// generates a signal build up by the specified function type. v1.4
// generates random signal (uniform, normal or chi-squared)

FUNCTION_BLOCK FB_FunctionGenerator
VAR_INPUT
	bEnable		: BOOL 	:= TRUE;
	fSamplingRate : LREAL := 10000.0; // in Hz
	nOversamples : UDINT := 10;
	fFrequency	: LREAL := 1000;	// in [Hz]
	fAmplitude	: LREAL := 1;
	fOffset		: LREAL	:= 0;	
	nDutyCycle	: UINT 	:= 50;		// % (for pulse function)
	nSeed		: INT	:= 1;	 
	aRange		: ARRAY [1..2] OF LREAL := [0,1];
	eRandType	: E_DistributionType	:= E_DistributionType.eNormal;
	eFunction	: E_FunctionType := E_FunctionType.eSine;	
END_VAR
VAR_OUTPUT
	bError		: BOOL;
	aSignal		: ARRAY[1..cOversamples] OF LREAL;
END_VAR
VAR
	bInit						: BOOL := TRUE;
	fLastSamplingRate : LREAL;
	nLastOversamples : UDINT;
	fLastFrequency				: LREAL;		// in [Hz]
	fLastAmplitude				: LREAL;
	fLastOffset					: LREAL;
	nLastDutyCycle				: UINT;
	eLastFunction				: E_FunctionType;
	
	nSamples					: UDINT;
	fCycleTime					: LREAL;		// in [s]
	fDelta						: LREAL;		// amplitude delta per sample
	fPhase						: LREAL;		// in [°]
	nSign						: INT := 1;		// 1 or -1
	fLastSignalValue			: LREAL;		// amplitude
	fPeriod						: LREAL;		// in [s]
	fAngularIncrement			: LREAL;		// in [°]
	fAngularIncrementPerCycle	: LREAL;		// in [°]
	fAngularIncrementPerSample	: LREAL;		// in [°]
	(* for modulated signal *)
	fCarrierFrequency			: LREAL := 500;	// in [Hz] (sine)
	fCarrierAmplitude			: LREAL := 1;
	fCarrierPeriod				: LREAL;		// in [s]
	fCarrierAngularIncrement			: LREAL;		// in [°]
	fCarrierAngularIncrementPerCycle	: LREAL;		// in [°]
	fCarrierAngularIncrementPerSample	: LREAL;		// in [°]
	
	fbDrand						: ARRAY[1..cOversamples] OF DRAND;		
	bNormalDist					: BOOL := TRUE;
	
	fY1							: LREAL;
	fY2							: LREAL;
	fX1							: LREAL;
	fX2							: LREAL;
	
	fbRAND1						: DRAND;
	fbRAND2						: DRAND;				
END_VAR

IF bEnable THEN

	IF fLastSamplingRate <> fSamplingRate THEN
		bInit := TRUE; // For automatic initializing
		fLastSamplingRate := fSamplingRate;
	END_IF
	IF nLastOversamples <> nOversamples THEN
		bInit := TRUE; // For automatic initializing
		nLastOversamples := nOversamples;
	END_IF
	
	IF fLastFrequency <> fFrequency THEN
		bInit := TRUE; // For automatic initializing
		fLastFrequency := fFrequency;
	END_IF
	IF fLastAmplitude <> fAmplitude THEN
		bInit := TRUE; // For automatic initializing
		fLastAmplitude := fAmplitude;
	END_IF
	IF fLastOffset <> fOffset THEN
		bInit := TRUE; // For automatic initializing
		fLastOffset := fOffset;
	END_IF
	IF nLastDutyCycle <> nDutyCycle THEN
		bInit := TRUE; // For automatic initializing
		nLastDutyCycle := nDutyCycle;
	END_IF
	IF eLastFunction <> eFunction THEN
		bInit := TRUE; // For automatic initializing
		eLastFunction := eFunction;
	END_IF
	IF bInit THEN
		// Get taks info	
//		fbGetTaskIdx();
//		fCycleTime := TwinCAT_SystemInfoVarList._TaskInfo[fbGetTaskIdx.index].CycleTime (*100ns*) / (10.0 * 1000.0 * 1000.0);	
		fCycleTime	 := nOversamples/fSamplingRate;
		fLastSignalValue := 0;
		nSign := 1;
		fAngularIncrement := 0;
		// Flush out old data
		MEMSET(ADR(aSignal), 0, SIZEOF(aSignal));
		IF fFrequency <> 0 AND fCycleTime > 0 THEN		
			// Calculate period, increments per plc cycle, increment per oversample
			IF cOversamples <> 0 THEN			
				IF eFunction = E_FunctionType.eSine THEN
					fPeriod := 1/fFrequency;
					fAngularIncrementPerCycle := 360*(fCycleTime/fPeriod);
					fAngularIncrementPerSample := fAngularIncrementPerCycle/cOversamples;
					// no phase adjustment
					bInit := FALSE;
				ELSIF eFunction = E_FunctionType.eConst	THEN
					bInit := FALSE;	
				ELSIF eFunction = E_FunctionType.eSquare	THEN
					fPeriod := 1/fFrequency;
					fAngularIncrementPerCycle := 360*(fCycleTime/fPeriod);
					fAngularIncrementPerSample := fAngularIncrementPerCycle/cOversamples;
					fPhase := 0.5*360;
					bInit := FALSE;
				ELSIF eFunction = E_FunctionType.ePulse THEN
					fPeriod := 1/fFrequency;
					fAngularIncrementPerCycle := 360*(fCycleTime/fPeriod);
					fAngularIncrementPerSample := fAngularIncrementPerCycle/cOversamples;
					IF nDutyCycle > 100 THEN
						nDutyCycle := 100;
					END_IF
					fPhase := (UDINT_TO_LREAL(nDutyCycle)/100)*360;
					bInit := FALSE;					
				ELSIF eFunction = E_FunctionType.eTriangular THEN
					fPeriod := 1/fFrequency;				
					fAngularIncrementPerCycle := 360*(fCycleTime/fPeriod);
					fAngularIncrementPerSample := fAngularIncrementPerCycle/cOversamples;
					fPhase := 0.5*360; 
					fDelta := 4*(fAmplitude/(360/fAngularIncrementPerSample));				
					bInit := FALSE;
				ELSIF eFunction = E_FunctionType.eTrapezoid THEN
					fPeriod := 1/fFrequency;				
					fAngularIncrementPerCycle := 360*(fCycleTime/fPeriod);
					fAngularIncrementPerSample := fAngularIncrementPerCycle/cOversamples;
					fPhase := 0.5*360; 
					fDelta := 4*(fAmplitude/(360/fAngularIncrementPerSample));				
					bInit := FALSE;					
				ELSIF eFunction = E_FunctionType.eSawtooth THEN
					fPeriod := 1/fFrequency;			
					fAngularIncrementPerCycle := 360*(fCycleTime/fPeriod);		
					fAngularIncrementPerSample := fAngularIncrementPerCycle/cOversamples;
					fDelta := fAmplitude/(360/fAngularIncrementPerSample);
					bInit := FALSE;
				ELSIF eFunction = E_FunctionType.eAM THEN
					fPeriod := 1/fFrequency;
					fAngularIncrementPerCycle := 360*(fCycleTime/fPeriod);
					fAngularIncrementPerSample := fAngularIncrementPerCycle/cOversamples;
					// no phase adjustment
					fCarrierPeriod := 1/fCarrierFrequency;
					fCarrierAngularIncrementPerCycle := 360*(fCycleTime/fCarrierPeriod);
					fCarrierAngularIncrementPerSample := fCarrierAngularIncrementPerCycle/cOversamples;				
					// no phase adjustment	
					bInit := FALSE;			
				ELSIF eFunction = E_FunctionType.eRand THEN	
					fbRAND1(Seed := nSeed);
					fbRAND2(Seed := nSeed+1);
					bInit := FALSE;
				ELSE
					bError := TRUE;	
				END_IF
			ELSE
				bError := TRUE;
			END_IF
		ELSE
			bError := TRUE;
		END_IF
	END_IF
	
	// Enable function generator
	IF NOT bError THEN		
		CASE eFunction OF		
			// const: constant signal
			E_FunctionType.eConst: Const();
			
			// sine: typical for vibrations originating from rotating machine
			E_FunctionType.eSine: Sine();			
			
			// square: mixed sine signals good for analyzing spectrum				
			E_FunctionType.eSquare: Square();
			
			// pulse: mixed sine signals good for analyzing spectrum				
			E_FunctionType.ePulse: Pulse();
	
			// sawtooth: ramp-type vibrations, continuously increasing			
			E_FunctionType.eSawtooth: Sawtooth();
		
			// triangular: mixed sine signals good for analyzing spectrum
			E_FunctionType.eTriangular: Triangular();
			
			// Trapezoid: trapezoid signal
			E_FunctionType.eTrapezoid: Trapezoid();
		
			// amplitude modulation: typical for vibrations originating from gear-tooth failure or bearing faults
			// Carrier signal with own frequency and amplitude		
			E_FunctionType.eAM: AM();	

			// random nosie: typical for disturbance signal				
		END_CASE
	END_IF
ELSE
	// Flush out old data
	MEMSET(ADR(aSignal), 0, SIZEOF(aSignal));
END_IF

METHOD PUBLIC AddAbsoluteNoise
VAR_INPUT
	fAbsoluteNoise	: LREAL;
END_VAR
VAR_IN_OUT
	aSignal		: ARRAY[1..cOversamples] OF LREAL;
END_VAR
VAR
	fNoise :LREAL;
END_VAR
FOR nSamples := 1 TO cOversamples DO	
	fbRAND1(Num => fNoise); // betwenn 0-1
	fNoise:= (fNoise*2 -1.0) * fAbsoluteNoise;
	aSignal[nSamples] := aSignal[nSamples] + fNoise;
END_FOR
END_METHOD

METHOD PRIVATE AM
VAR_INPUT
END_VAR
FOR nSamples := 1 TO cOversamples DO
	// base signal * carrier signal
	aSignal[nSamples] := ( fAmplitude*SIN(2*PI*(fAngularIncrement+(nSamples-1)*fAngularIncrementPerSample)/360) + fOffset )
							* ( fCarrierAmplitude*SIN(2*PI*(fCarrierAngularIncrement+(nSamples-1)*fCarrierAngularIncrementPerSample)/360) );
END_FOR
// Increment angular positions
fAngularIncrement := fAngularIncrement + fAngularIncrementPerCycle;
fCarrierAngularIncrement := fCarrierAngularIncrement + fCarrierAngularIncrementPerCycle;
END_METHOD

METHOD PRIVATE Const
VAR_INPUT
END_VAR
FOR nSamples := 1 TO cOversamples DO
	
	aSignal[nSamples] := fAmplitude;
	
	aSignal[nSamples] := aSignal[nSamples] + fOffset;
END_FOR
END_METHOD

METHOD PRIVATE Pulse
VAR_INPUT
END_VAR
FOR nSamples := 1 TO cOversamples DO
	// For pulse wave (unequal phases)
	IF (fAngularIncrement >= 360) THEN
		fAngularIncrement := fAngularIncrement - DINT_TO_LREAL(LREAL_TO_DINT(fAngularIncrement/360))*360;
		// or with Tc2_Math library: fAngularIncrement := LMOD(fAngularIncrement,360);
	END_IF
	IF (fAngularIncrement < fPhase) THEN
		nSign := 1;		
	ELSIF (fAngularIncrement >= fPhase) THEN
		nSign := 0;
	END_IF
	fAngularIncrement := fAngularIncrement + fAngularIncrementPerSample;
	
	aSignal[nSamples] := nSign*fAmplitude;
	
	aSignal[nSamples] := aSignal[nSamples] + fOffset;
END_FOR
END_METHOD

METHOD PRIVATE Sawtooth
VAR_INPUT
END_VAR
FOR nSamples := 1 TO cOversamples DO
	// For sawtooth wave (equal phase = period/2)
	IF (fAngularIncrement >= 360) THEN
		fAngularIncrement := fAngularIncrement - DINT_TO_LREAL(LREAL_TO_DINT(fAngularIncrement/360))*360;
		// or with Tc2_Math library: fAngularIncrement := LMOD(fAngularIncrement,360);
		fLastSignalValue := fLastSignalValue -fAmplitude;
	END_IF
	fAngularIncrement := fAngularIncrement + fAngularIncrementPerSample;

	aSignal[nSamples] := fLastSignalValue + fDelta;

	// Store last sample
	fLastSignalValue := aSignal[nSamples];
	
	aSignal[nSamples] := aSignal[nSamples] + fOffset;					
END_FOR
END_METHOD

METHOD PRIVATE Sine
VAR_INPUT
END_VAR
FOR nSamples := 1 TO cOversamples DO
	aSignal[nSamples] := fAmplitude*SIN(2*PI*(fAngularIncrement+(nSamples-1)*fAngularIncrementPerSample)/360);

	aSignal[nSamples] := aSignal[nSamples] + fOffset;
END_FOR

// Increment angular position
fAngularIncrement := fAngularIncrement + fAngularIncrementPerCycle;
END_METHOD

METHOD PRIVATE Square
VAR_INPUT
END_VAR
FOR nSamples := 1 TO cOversamples DO
	// For square wave (equal phase = period/2)
	IF (fAngularIncrement >= 360) THEN
		fAngularIncrement := fAngularIncrement - DINT_TO_LREAL(LREAL_TO_DINT(fAngularIncrement/360))*360;
		// or with Tc2_Math library: fAngularIncrement := LMOD(fAngularIncrement,360);
	END_IF
	IF (fAngularIncrement < fPhase) THEN
		nSign := 1;
	ELSIF (fAngularIncrement >= fPhase) THEN
		nSign := -1;
	END_IF
	fAngularIncrement := fAngularIncrement + fAngularIncrementPerSample;
	
	aSignal[nSamples] := nSign*fAmplitude;
	
	aSignal[nSamples] := aSignal[nSamples] + fOffset;
END_FOR
END_METHOD

METHOD PRIVATE Trapezoid
VAR_INPUT
END_VAR
FOR nSamples := 1 TO cOversamples DO
	IF (fAngularIncrement >= 360) THEN
		fAngularIncrement := fAngularIncrement - DINT_TO_LREAL(LREAL_TO_DINT(fAngularIncrement/360))*360;
		// or with Tc2_Math library: fAngularIncrement := LMOD(fAngularIncrement,360);
	END_IF
	// Negative delta -> Positive delta
	IF fAngularIncrement < fPhase/2 THEN	
		nSign := 1;		
	ELSIF fAngularIncrement >= fPhase/2 AND fAngularIncrement < fPhase THEN
		nSign := -1;
	ELSIF fAngularIncrement >= fPhase THEN
		nSign := 0;	
	END_IF
	fAngularIncrement := fAngularIncrement + fAngularIncrementPerSample;
	
	aSignal[nSamples] := fLastSignalValue + nSign*fDelta;
	IF aSignal[nSamples] > fAmplitude THEN
		aSignal[nSamples] := aSignal[nSamples] - 2*(aSignal[nSamples]-fAmplitude);
	ELSIF aSignal[nSamples] < (-1)*fAmplitude THEN
		aSignal[nSamples] := aSignal[nSamples] - 2*(aSignal[nSamples]+fAmplitude);
	END_IF
	
	// Store last sample
	fLastSignalValue := aSignal[nSamples];		
	
	IF fLastSignalValue > fAmplitude * 0.5 THEN
		aSignal[nSamples] := fAmplitude * 0.5;
	END_IF
	
	aSignal[nSamples] := aSignal[nSamples] + fOffset;
END_FOR
END_METHOD

METHOD PRIVATE Triangular
VAR_INPUT
END_VAR
FOR nSamples := 1 TO cOversamples DO
	IF (fAngularIncrement >= 360) THEN
		fAngularIncrement := fAngularIncrement - DINT_TO_LREAL(LREAL_TO_DINT(fAngularIncrement/360))*360;
		// or with Tc2_Math library: fAngularIncrement := LMOD(fAngularIncrement,360);
	END_IF
	// Negative delta -> Positive delta
	IF fAngularIncrement < fPhase/2 THEN	
		nSign := 1;		
	ELSIF fAngularIncrement >= fPhase/2 AND fAngularIncrement < 3*fPhase/2 THEN
		nSign := -1;
	ELSIF fAngularIncrement >= 3*fPhase/2 THEN
		nSign := 1;	
	END_IF
	fAngularIncrement := fAngularIncrement + fAngularIncrementPerSample;
	
	aSignal[nSamples] := fLastSignalValue + nSign*fDelta;
	IF aSignal[nSamples] > fAmplitude THEN
		aSignal[nSamples] := aSignal[nSamples] - 2*(aSignal[nSamples]-fAmplitude);
	ELSIF aSignal[nSamples] < (-1)*fAmplitude THEN
		aSignal[nSamples] := aSignal[nSamples] - 2*(aSignal[nSamples]+fAmplitude);
	END_IF
	
	// Store last sample
	fLastSignalValue := aSignal[nSamples];		
	
	aSignal[nSamples] := aSignal[nSamples] + fOffset;
END_FOR
END_METHOD

END_FUNCTION_BLOCK

(* stored: Version 1.1.0.1, ProductVersion 3.1.4024.12
   POU FB_FunctionGenerator: Id {69c9f199-36dd-4eeb-9032-3058e23f3e10}, SpecialFunc None
   Method AddAbsoluteNoise: Id {7b96f9f0-18f5-40f1-8831-de6c91807439}
   Method AM: Id {72cbf823-a283-4d76-abbd-04bdf01b5b09}
   Method Const: Id {579094e5-092b-45b5-b05e-82e1b2eb2d91}
   Method Pulse: Id {589d36d2-806a-469d-be67-d4a57f34ac9b}
   Method Sawtooth: Id {8523d13a-521d-4b1f-b20c-157f6fbf4477}
   Method Sine: Id {3cbb271a-9c9c-458c-97e2-003c0bd11c99}
   Method Square: Id {782e04ad-12e1-4b0e-9ce3-b0830baab1f6}
   Method Trapezoid: Id {440568a5-7a01-47a2-b38d-7686581ec158}
   Method Triangular: Id {6fd33f65-9406-482d-8e99-c66fd3f34453} *)
